# B&R Automation Studio project Lib_IecFrmtStr
Automation Studio 4.7.4.67 SP

## Configuration ARsim

### Task classes (Cpu.sw)
```
Cyclic#1 (cycle 1000 us, tolerance 0 us):
  Program <- Program.prg
Binaries: FWRules, TCData, udbdef, asfw, User, iomap, sysconf, arconfig, ashwd, Role, ashwac
Libraries: BRSE_ARL, AsBrStr, ArEventLog, sys_lib, runtime, asieccon, astime
```

### Hardware
```
PC : PC_any v1.1.0.0 (OrderNumber=PC)
  ConfigurationID = Lib_IecFrmtStr_ARsim
  SystemTick = 1000
  Cyclic1Duration = 1000
  Cyclic1Tolerance = 0
```

## Logical view

Binary libraries used (declarations not repeated): operator, runtime, astime, AsIecCon, BRSE_ARL, AsBrStr, ArEventLog, sys_lib


### Program Logical/Program (IEC)

#### Variables.var
```iecst
VAR
	AllocationReturnStatus : UDINT;
	CyclicReturnStatus : UDINT;
	FreeReturnStatus : UDINT;
END_VAR
VAR CONSTANT
	STR_LEN_ALARM_MSG : USINT := 125;
END_VAR
```

#### Main.st
```iecst
(*******************************************************************************
 * Copyright: B&R Industrial Automation
 * Author:    Tyler Matijevich
 * Created:   September 27, 2020/11:19
********************************************************************************
 * Description: Example program for formatting string in IEC code and logging
 user entries in the logger
********************************************************************************)

PROGRAM _INIT

	// Allocates the FIFO buffer for the logger
	AllocationReturnStatus := BRSE_ARL_Alloc(ID := 1, Name := 'AppLog', LogbookSize := 10000, MessageSize := STR_LEN_ALARM_MSG, BufferedEntries := 25);

END_PROGRAM

PROGRAM _CYCLIC

	// Flush pending entries to the logbook
	CyclicReturnStatus := BRSE_ARL_Cyclic(ID := 1);

END_PROGRAM

PROGRAM _EXIT

	// Deallocate the FIFO buffer
	FreeReturnStatus := BRSE_ARL_Free(ID := 1);

END_PROGRAM
```

Listed in the project but not available here: Logical/Global.typ, Logical/Global.var
